// TIA Portal V20 export
FUNCTION_BLOCK "定位轴基本控制"   // FB1, LAD
{ S7_Optimized_Access := 'TRUE' }
// stored: MemoryReserve 100, SetENOAutomatically false
   VAR_INPUT
      轴号 : TO_PositioningAxis;
      使能 : Bool;
      回原 : Bool;
      回原模式 : Int;
      绝对定位 : Bool;
      相对定位 : Bool;
      暂停 : Bool;
      复位 : Bool;
      绝对位置 : Real;
      绝对速度 : Real;
      相对位置 : Real;
      相对速度 : Real;
      点动正转 : Bool;
      点动反转 : Bool;
      点动速度 : Real;
   END_VAR
   VAR_OUTPUT
      轴已启用 : Bool;
      使能错误 : Bool;
      回原完成 : Bool;
      回原错误 : Bool;
      绝对定位完成 : Bool;
      绝对定位错误 : Bool;
      相对定位完成 : Bool;
      相对定位错误 : Bool;
      点动中 : Bool;
      点动错误 : Bool;
      当前位置 : LReal;
      当前速度 : LReal;
   END_VAR
   VAR
      MC_Power_Instance { S7_SetPoint := 'True'} : MC_POWER;
      MC_Home_Instance { S7_SetPoint := 'True'} : MC_HOME;
      MC_MoveAbsolute_Instance { S7_SetPoint := 'True'} : MC_MOVEABSOLUTE;
      MC_MoveRelative_Instance { S7_SetPoint := 'True'} : MC_MOVERELATIVE;
      MC_Reset_Instance { S7_SetPoint := 'True'} : MC_RESET;
      MC_Halt_Instance { S7_SetPoint := 'True'} : MC_HALT;
      MC_MoveJog_Instance { S7_SetPoint := 'True'} : MC_MOVEJOG;
   END_VAR
   VAR_TEMP
      复位完成 : Bool;
      复位错误 : Bool;
      暂停完成 : Bool;
      暂停错误 : Bool;
   END_VAR
   VAR_TEMP   // added for the SCL form of the ladder/FBD networks
      _w1 : Bool;
      _w2 : Bool;
      _w3 : Bool;
   END_VAR
BEGIN

REGION Network 1
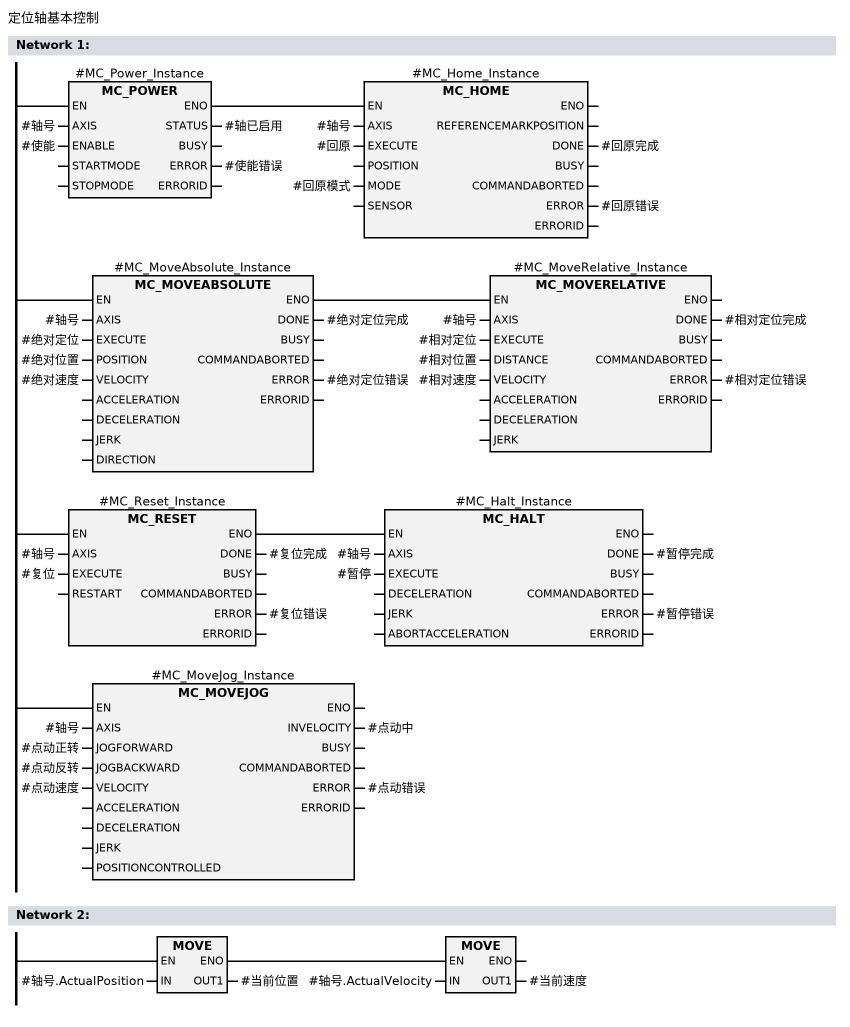
   RUNG wire#powerrail
      #MC_Power_Instance.MC_POWER(Axis := #轴号, Enable := #使能, StartMode :=, StopMode :=, Status => #轴已启用, Busy =>, Error => #使能错误, ErrorId =>)
      #MC_Home_Instance.MC_HOME(Axis := #轴号, Execute := #回原, Position :=, Mode := #回原模式, Sensor :=, ReferenceMarkPosition =>, Done => #回原完成, Busy =>, CommandAborted =>, Error => #回原错误, ErrorId =>)
   END_RUNG
   RUNG wire#powerrail
      #MC_MoveAbsolute_Instance.MC_MOVEABSOLUTE(Axis := #轴号, Execute := #绝对定位, Position := #绝对位置, Velocity := #绝对速度, Acceleration :=, Deceleration :=, Jerk :=, Direction :=, Done => #绝对定位完成, Busy =>, CommandAborted =>, Error => #绝对定位错误, ErrorId =>)
      #MC_MoveRelative_Instance.MC_MOVERELATIVE(Axis := #轴号, Execute := #相对定位, Distance := #相对位置, Velocity := #相对速度, Acceleration :=, Deceleration :=, Jerk :=, Done => #相对定位完成, Busy =>, CommandAborted =>, Error => #相对定位错误, ErrorId =>)
   END_RUNG
   RUNG wire#powerrail
      #MC_Reset_Instance.MC_RESET(Axis := #轴号, Execute := #复位, Restart :=, Done => #复位完成, Busy =>, CommandAborted =>, Error => #复位错误, ErrorId =>)
      #MC_Halt_Instance.MC_HALT(Axis := #轴号, Execute := #暂停, Deceleration :=, Jerk :=, AbortAcceleration :=, Done => #暂停完成, Busy =>, CommandAborted =>, Error => #暂停错误, ErrorId =>)
   END_RUNG
   RUNG wire#powerrail
      #MC_MoveJog_Instance.MC_MOVEJOG(Axis := #轴号, JogForward := #点动正转, JogBackward := #点动反转, Velocity := #点动速度, Acceleration :=, Deceleration :=, Jerk :=, PositionControlled :=, InVelocity => #点动中, Busy =>, CommandAborted =>, Error => #点动错误, ErrorId =>)
   END_RUNG
   // the same network as SCL:
   #MC_Power_Instance(Axis := #轴号, Enable := #使能, Status => #轴已启用, Error => #使能错误, ENO => #_w1);   // MC_POWER
   IF #_w1 THEN
       #MC_Home_Instance(Axis := #轴号, Execute := #回原, Mode := #回原模式, Done => #回原完成, Error => #回原错误);   // MC_HOME
   END_IF;
   #MC_MoveAbsolute_Instance(Axis := #轴号,   // MC_MOVEABSOLUTE
                           Execute := #绝对定位,
                           Position := #绝对位置,
                           Velocity := #绝对速度,
                           Done => #绝对定位完成,
                           Error => #绝对定位错误,
                           ENO => #_w2);
   IF #_w2 THEN
       #MC_MoveRelative_Instance(Axis := #轴号,   // MC_MOVERELATIVE
                               Execute := #相对定位,
                               Distance := #相对位置,
                               Velocity := #相对速度,
                               Done => #相对定位完成,
                               Error => #相对定位错误);
   END_IF;
   #MC_Reset_Instance(Axis := #轴号, Execute := #复位, Done => #复位完成, Error => #复位错误, ENO => #_w3);   // MC_RESET
   IF #_w3 THEN
       #MC_Halt_Instance(Axis := #轴号, Execute := #暂停, Done => #暂停完成, Error => #暂停错误);   // MC_HALT
   END_IF;
   #MC_MoveJog_Instance(Axis := #轴号,   // MC_MOVEJOG
                        JogForward := #点动正转,
                        JogBackward := #点动反转,
                        Velocity := #点动速度,
                        InVelocity => #点动中,
                        Error => #点动错误);
END_REGION

REGION Network 2
   RUNG wire#powerrail
      Move(in := #轴号.ActualPosition, out1 => #当前位置)
      Move(in := #轴号.ActualVelocity, out1 => #当前速度)
   END_RUNG
   // the same network as SCL:
   #当前位置 := #轴号.ActualPosition;
   #当前速度 := #轴号.ActualVelocity;
END_REGION
END_FUNCTION_BLOCK
